// TIA Portal project "practica_6" (V15)

(* hardware
DEVICE "PC-Scada"  SIMATIC PC station
   slot 0: "Estación PC SIMATIC"  Rail  SIMATIC PC-Station  V1.0
      slot 125: "Stationmanager"  Station_Manager  V6.0.4
   slot 1: "HMI_RT_1"  WinCC RT Advanced  6AV2 104-0xxxx-xxxx  15.0.0.0
      slot 33792: "Interfaz host"  Host interface
   slot 2: "IE general_1"  IE General  IE_CP  V8.2.0
DEVICE "S7-1200 station_1"  S7-1200 Station
   slot 0: "Rack_0"  S7-1200 Rack  Rack  V1.0
   slot 1: "PLC_1"  CPU 1215C AC/DC/Rly  6ES7 215-1BG40-0XB0  V4.2
*)

// ===== PLC "PLC_1"  CPU 1215C AC/DC/Rly =====

VAR_GLOBAL   // PLC tag table "Tabla de variables_1"
   "B1" AT %I0.0 : Bool;
   "B2" AT %I0.1 : Bool;
   "S1" AT %I0.2 : Bool;
   "S2" AT %I0.3 : Bool;
   "V1" AT %Q0.4 : Bool;
   "V2" AT %Q0.5 : Bool;
   "E10" AT %M0.6 : Bool;
   "E11" AT %M0.7 : Bool;
   "E21" AT %M1.0 : Bool;
   "E20" AT %M1.1 : Bool;
   "E30" AT %M1.2 : Bool;
   "P1" AT %Q1.3 : Bool;
   "P2" AT %Q1.4 : Bool;
   "M" AT %Q1.5 : Bool;
   "E0" AT %M1.6 : Bool;
END_VAR

FUNCTION "Acciones" : Void   // FC1, LAD
{ S7_Optimized_Access := 'TRUE' }
VERSION : 0.1
BEGIN

REGION Network 1
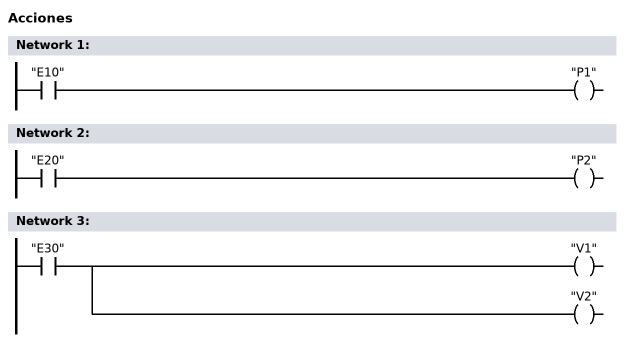
   RUNG wire#powerrail
      Contact( "E10" )
      Coil( "P1" )
   END_RUNG
   // the same network as SCL:
   "P1" := "E10";
END_REGION

REGION Network 2
   RUNG wire#powerrail
      Contact( "E20" )
      Coil( "P2" )
   END_RUNG
   // the same network as SCL:
   "P2" := "E20";
END_REGION

REGION Network 3
   RUNG wire#powerrail
      Contact( "E30" )
      wire#w1
      Coil( "V1" )
   END_RUNG
   RUNG wire#w1
      Coil( "V2" )
   END_RUNG
   // the same network as SCL:
   "V1" := "E30";
   "V2" := "E30";
END_REGION
END_FUNCTION

FUNCTION "Principal" : Void   // FC2, LAD
{ S7_Optimized_Access := 'TRUE' }
VERSION : 0.1
BEGIN

REGION Network 1
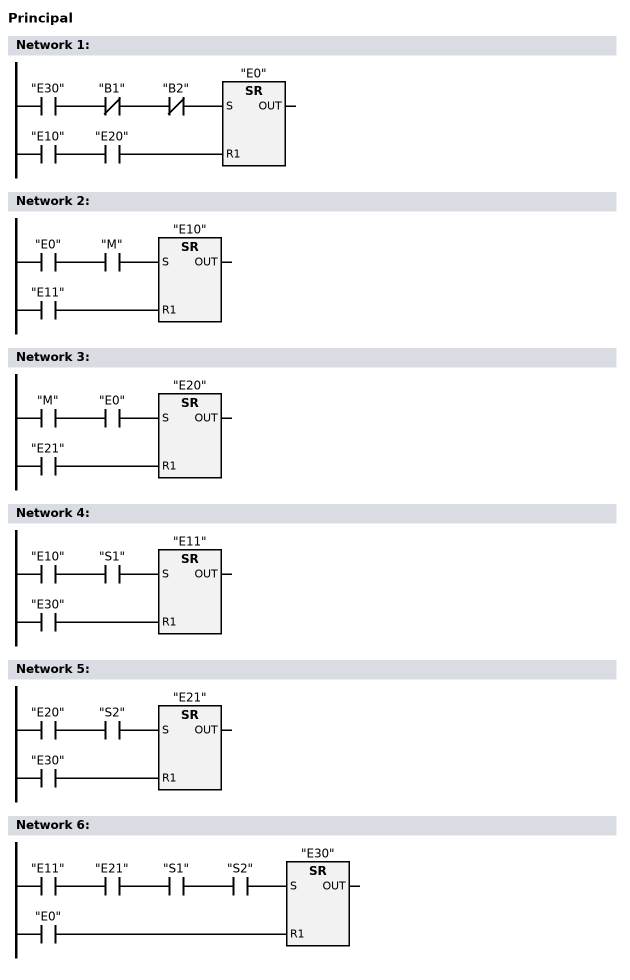
   RUNG wire#powerrail
      Contact( "E30" )
      I_Contact( "B1" )
      I_Contact( "B2" )
      S_SR(operand := "E0", r1 := wire#w1)
   END_RUNG
   RUNG wire#powerrail
      Contact( "E10" )
      Contact( "E20" )
   END_RUNG wire#w1
   // the same network as SCL:
   IF "E30" AND NOT "B1" AND NOT "B2" THEN
       "E0" := TRUE;   // SR flip-flop
   END_IF;
   IF "E10" AND "E20" THEN "E0" := FALSE; END_IF;
END_REGION

REGION Network 2
   RUNG wire#powerrail
      Contact( "E0" )
      Contact( "M" )
      S_SR(operand := "E10", r1 := wire#w1)
   END_RUNG
   RUNG wire#powerrail
      Contact( "E11" )
   END_RUNG wire#w1
   // the same network as SCL:
   IF "E0" AND "M" THEN
       "E10" := TRUE;   // SR flip-flop
   END_IF;
   IF "E11" THEN "E10" := FALSE; END_IF;
END_REGION

REGION Network 3
   RUNG wire#powerrail
      Contact( "M" )
      Contact( "E0" )
      S_SR(operand := "E20", r1 := wire#w1)
   END_RUNG
   RUNG wire#powerrail
      Contact( "E21" )
   END_RUNG wire#w1
   // the same network as SCL:
   IF "M" AND "E0" THEN
       "E20" := TRUE;   // SR flip-flop
   END_IF;
   IF "E21" THEN "E20" := FALSE; END_IF;
END_REGION

REGION Network 4
   RUNG wire#powerrail
      Contact( "E10" )
      Contact( "S1" )
      S_SR(operand := "E11", r1 := wire#w1)
   END_RUNG
   RUNG wire#powerrail
      Contact( "E30" )
   END_RUNG wire#w1
   // the same network as SCL:
   IF "E10" AND "S1" THEN
       "E11" := TRUE;   // SR flip-flop
   END_IF;
   IF "E30" THEN "E11" := FALSE; END_IF;
END_REGION

REGION Network 5
   RUNG wire#powerrail
      Contact( "E20" )
      Contact( "S2" )
      S_SR(operand := "E21", r1 := wire#w1)
   END_RUNG
   RUNG wire#powerrail
      Contact( "E30" )
   END_RUNG wire#w1
   // the same network as SCL:
   IF "E20" AND "S2" THEN
       "E21" := TRUE;   // SR flip-flop
   END_IF;
   IF "E30" THEN "E21" := FALSE; END_IF;
END_REGION

REGION Network 6
   RUNG wire#powerrail
      Contact( "E11" )
      Contact( "E21" )
      Contact( "S1" )
      Contact( "S2" )
      S_SR(operand := "E30", r1 := wire#w1)
   END_RUNG
   RUNG wire#powerrail
      Contact( "E0" )
   END_RUNG wire#w1
   // the same network as SCL:
   IF "E11" AND "E21" AND "S1" AND "S2" THEN
       "E30" := TRUE;   // SR flip-flop
   END_IF;
   IF "E0" THEN "E30" := FALSE; END_IF;
END_REGION
END_FUNCTION

ORGANIZATION_BLOCK "Main"   // OB1, LAD, ProgramCycle
TITLE = "Main Program Sweep (Cycle)"
{ S7_Optimized_Access := 'TRUE' }
VERSION : 0.1
   VAR_INPUT
      Initial_Call : Bool;   // Initial call of this OB
      Remanence : Bool;   // =True, if remanent data are available
   END_VAR
BEGIN

REGION Network 1
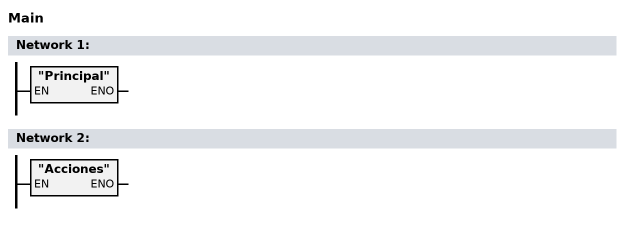
   RUNG wire#powerrail
      "Principal"()
   END_RUNG
   // the same network as SCL:
   "Principal"();
END_REGION

REGION Network 2
   RUNG wire#powerrail
      "Acciones"()
   END_RUNG
   // the same network as SCL:
   "Acciones"();
END_REGION
END_ORGANIZATION_BLOCK

ORGANIZATION_BLOCK "StartUp"   // OB123, LAD, ProgramCycle
TITLE = "Main Program Sweep (Cycle)"
{ S7_Optimized_Access := 'TRUE' }
VERSION : 0.1
   VAR_INPUT
      Initial_Call : Bool;   // Initial call of this OB
      Remanence : Bool;   // =True, if remanent data are available
   END_VAR
BEGIN

REGION Network 1
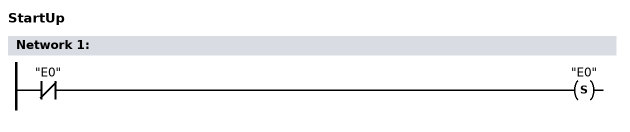
   RUNG wire#powerrail
      I_Contact( "E0" )
      S_Coil( "E0" )
   END_RUNG
   // the same network as SCL:
   IF NOT "E0" THEN "E0" := TRUE; END_IF;
END_REGION
END_ORGANIZATION_BLOCK

(* ===== HMI "HMI_RT_1" =====
connection "Conexión_1": ETHERNET, SIMATIC S7 300/400 MPI

screen "Imagen_projecto_6" 1024x768
   GraphicView "Visor de gráficos_1" at 0,0 size 1017x765; Picture "iStock-616891500-730x620"
   Button "Botón_1" at 55,107 size 220x88; TextOff 'INICIAR'
   GraphicView "Visor de gráficos_2" at 313,45 size 345x384; Picture "Gráfico_1"
   GraphicView "Visor de gráficos_3" at 660,47 size 336x381; Picture "Gráfico_1"
   GraphicView "Visor de gráficos_4" at 545,428 size 192x297; Picture "Gráfico_3"
   GraphicView "Visor de gráficos_5" at 65,508 size 292x233; Picture "Gráfico_5"
*)